{attribute 'strict'}
{attribute 'qualified_only'}
TYPE E_MachineMode :
(
	eUndefined				:= 0,
	eManual					:= 1,
	eMaintenance			:= 2,
	eAutomatic				:= 3,
	eSemiAutomatic			:= 4,
	eFirstFilling			:= 5,
	eEmptying				:= 6
);
END_TYPE

(* stored: Version 1.1.0.1, ProductVersion 3.1.4022.12
   DUT E_MachineMode: Id {a23e5493-84c3-4871-a5f6-ac2e3c5967dd} *)
